Yaskawa INFORM job: AAA.JBI

/JOB
//NAME AAA
//POS
///NPOS 2,0,0,0,0,0
///TOOL 9
///POSTYPE PULSE
///PULSE
C00000=-39381,59725,17195,7856,-45030,-8452
C00001=-5025,71334,30707,19220,-52923,-22152
//INST
///DATE 2023/03/01 22:04
///ATTR SC,RW
///GROUP1 RB1
NOP
MOVJ C00000 VJ=1.0
MOVL C00001 V=25.0 SRCH RIN#(3)=ON DIS=20.0
END
